FUNCTION_BLOCK ControlDescensoFin
VAR_INPUT
		SFCreset:BOOL;
	    SeguridadOK AT %I*: BOOL;
	    SensorArriba AT %I*: BOOL;
		SensorAbajo AT %I*:BOOL;
		Enabled AT %I*:BOOL;
		PuedeExtraer :BOOL;
		
		SensorPaletDentro AT %I*:BOOL;
		SensorPaletFuera AT %I*:BOOL;
		ElevadorLleno :BOOL;
		PulsadorBajar AT%I*: BOOL;
		PulsadorSubir AT%I*: BOOL;	

		PresenciaCintaArriba AT%I* :BOOL;
		PresenciaCintaAbajo AT %I* : BOOL;	
		
		ResetError :BOOL;
		
		MotorElevacion_Status AT%I*:UINT;
		MotorExtraccion_Status AT%I*:UINT;

END_VAR
VAR_OUTPUT
		MotorElevacion_Freq  AT%Q*: UINT;
	    MotorElevacion_Command AT%Q*: UINT;
		
		MotorExtraccion_Freq  AT%Q*: UINT;
	    MotorExtraccion_Command AT%Q*: UINT;
		
		Ready: BOOL; 
		
END_VAR
VAR
	VelocidadAlta :UINT := 4000;
	VelocidadBAJA :UINT := 1500;
	ModoVelocidadAlta :BOOL := FALSE;
	TiempoAltaVelocidad :TIME := T#3S;
	ERROR :BOOL;
	TimerEntradaSalida: TON;
	
	HomeOK :BOOL;
END_VAR

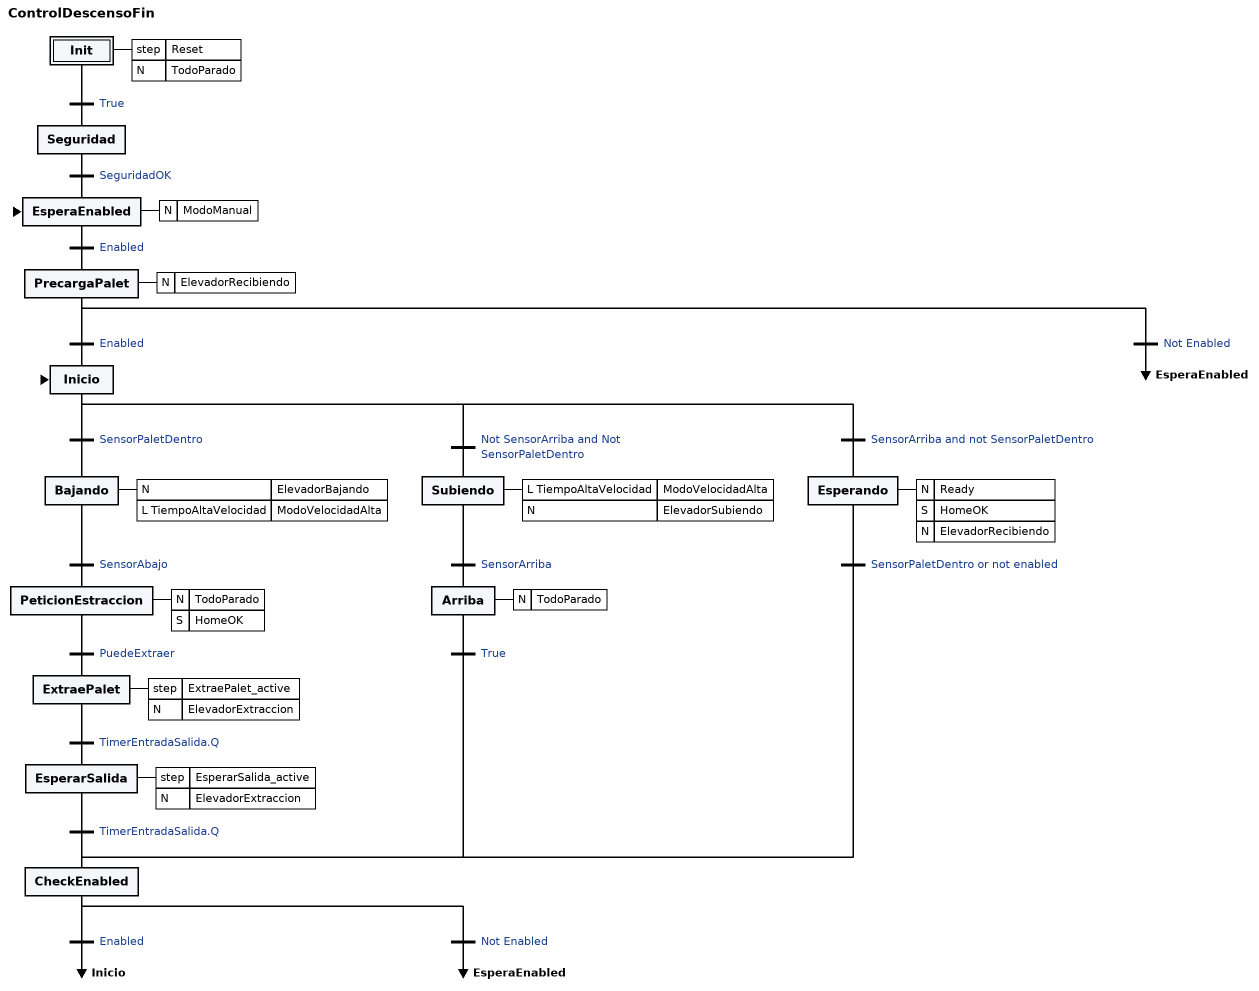
INITIAL_STEP Init:
    Reset(N);  // step action
    TodoParado(N);
END_STEP
TRANSITION FROM Init TO Seguridad
    := True;
END_TRANSITION
STEP Seguridad:
END_STEP
TRANSITION FROM Seguridad TO EsperaEnabled
    := SeguridadOK;
END_TRANSITION
STEP EsperaEnabled:
    ModoManual(N);
END_STEP
TRANSITION FROM EsperaEnabled TO PrecargaPalet
    := Enabled;
END_TRANSITION
STEP PrecargaPalet:  // min time T#2s
    ElevadorRecibiendo(N);
END_STEP
TRANSITION FROM PrecargaPalet TO Inicio
    := Enabled;
END_TRANSITION
TRANSITION FROM PrecargaPalet TO EsperaEnabled
    := Not Enabled;
END_TRANSITION
STEP Inicio:
END_STEP
TRANSITION FROM Inicio TO Bajando
    := SensorPaletDentro;
END_TRANSITION
STEP Bajando:
    ElevadorBajando(N);
    ModoVelocidadAlta(L, TiempoAltaVelocidad);
END_STEP
TRANSITION FROM Bajando TO PeticionEstraccion
    := SensorAbajo;
END_TRANSITION
STEP PeticionEstraccion:
    TodoParado(N);
    HomeOK(S);
END_STEP
TRANSITION FROM PeticionEstraccion TO ExtraePalet
    := PuedeExtraer;
END_TRANSITION
STEP ExtraePalet:  // min time T#1s
    ExtraePalet_active(N);  // step action
    ElevadorExtraccion(N);
END_STEP
TRANSITION FROM ExtraePalet TO EsperarSalida
    := TimerEntradaSalida.Q;
END_TRANSITION
STEP EsperarSalida:
    EsperarSalida_active(N);  // step action
    ElevadorExtraccion(N);
END_STEP
TRANSITION FROM EsperarSalida TO CheckEnabled
    := TimerEntradaSalida.Q;
END_TRANSITION
TRANSITION FROM Inicio TO Subiendo
    := Not SensorArriba and Not SensorPaletDentro;
END_TRANSITION
STEP Subiendo:
    ModoVelocidadAlta(L, TiempoAltaVelocidad);
    ElevadorSubiendo(N);
END_STEP
TRANSITION FROM Subiendo TO Arriba
    := SensorArriba;
END_TRANSITION
STEP Arriba:
    TodoParado(N);
END_STEP
TRANSITION FROM Arriba TO CheckEnabled
    := True;
END_TRANSITION
TRANSITION FROM Inicio TO Esperando
    := SensorArriba and not SensorPaletDentro;
END_TRANSITION
STEP Esperando:
    Ready(N);
    HomeOK(S);
    ElevadorRecibiendo(N);
END_STEP
TRANSITION FROM Esperando TO CheckEnabled
    := SensorPaletDentro or not enabled;
END_TRANSITION
STEP CheckEnabled:
END_STEP
TRANSITION FROM CheckEnabled TO Inicio
    := Enabled;
END_TRANSITION
TRANSITION FROM CheckEnabled TO EsperaEnabled
    := Not Enabled;
END_TRANSITION

ACTION ElevadorBajando:
MotorElevador(2);
MotorExtraccion(0);
END_ACTION

ACTION ElevadorExtraccion:

IF PuedeExtraer THEN
	MotorExtraccion(1);
ELSE 
	MotorExtraccion(0);
END_IF
END_ACTION

ACTION ElevadorRecibiendo:
MotorElevador(0);

IF Enabled THEN
	MotorExtraccion(2);
ELSE 
	MotorExtraccion(0);
END_IF
END_ACTION

ACTION ElevadorSubiendo:
MotorElevador(1);
MotorExtraccion(0);
END_ACTION

ACTION EsperarSalida_active:
TimerEntradaSalida(IN:=NOT PresenciaCintaAbajo, PT:= T#1S);
END_ACTION

ACTION ExtraePalet_active:
TimerEntradaSalida(IN:=PresenciaCintaAbajo, PT:= T#1S);
END_ACTION

ACTION ModoManual:


IF PulsadorSubir THEN
	MotorElevador(1);
		HomeOK :=FALSE;
ELSIF PulsadorBajar THEN
	MotorElevador(2);
		HomeOK :=FALSE;
ELSE
	MotorElevador(0);
END_IF
END_ACTION

METHOD PRIVATE MotorElevador : BOOL
VAR_INPUT
	Direccion : INT; //0 parado 1 subir 2 bajar
END_VAR
IF ModoVelocidadAlta AND HomeOK THEN
	MotorElevacion_Freq := 5000;
ELSE
	MotorElevacion_Freq := 1000;
END_IF


MotorElevacion_Command := 0;
MotorElevacion_Command.7 := 1 ; //Control Word Active

IF Direccion = 0 THEN
	MotorElevacion_Command.3 := 1 ; // Stop according to parameter setting	
ELSIF PresenciaCintaArriba OR PresenciaCintaAbajo THEN
	//ERROR: intenta mover elevador con obstatuclos
	//DEBE MOStrar error
	MotorElevacion_Command.3 := 1 ; // Stop according to parameter setting	
	
ELSIF Direccion  = 1 THEN
		
		MotorElevacion_Command.2 := 0 ; //1 reversed 0 fordward
		MotorElevacion_Command.0 := 1 ; // Run Command active
		HomeOK :=FALSE;

ELSIF Direccion= 2 THEN
	MotorElevacion_Command.2 := 1 ; //1 reversed 0 fordward
	MotorElevacion_Command.0 := 1 ; // Run Command active
		HomeOK :=FALSE;
ELSE
	MotorElevacion_Command.3 := 1 ; // Stop according to parameter setting	
END_IF
END_METHOD

METHOD PRIVATE MotorExtraccion : BOOL
VAR_INPUT
	Direccion : INT; //0 parado 1 salida 2 entrada
END_VAR

MotorExtraccion_Freq := gvl.VelocidadCinta * 100;
MotorExtraccion_Command := 0;
MotorExtraccion_Command.7 := 1 ; //Control Word Active

IF Direccion  = 1 THEN
	MotorExtraccion_Command.2 := 1 ; //1 reversed 0 fordward
	MotorExtraccion_Command.0 := 1 ; // Run Command active
ELSIF Direccion= 2 THEN
	MotorExtraccion_Command.2 := 0 ; //1 reversed 0 fordward
	MotorExtraccion_Command.0 := 1 ; // Run Command active
ELSE
	MotorExtraccion_Command.3 := 1 ; // Stop according to parameter setting	
END_IF
END_METHOD

ACTION RealizaHome:
MotorElevador(1);
MotorExtraccion(0);
END_ACTION

ACTION Reset:
HomeOK := FALSE;
SFCreset:=FALSE;
END_ACTION

ACTION TodoParado:
MotorElevador(0);
MotorExtraccion(0);
END_ACTION

END_FUNCTION_BLOCK

(* stored: Version 1.1.0.1, ProductVersion 3.1.4024.3
   POU ControlDescensoFin: Id {d10a53bb-d051-4ece-977c-1063e3a0bb26}, SpecialFunc None
   Action ElevadorBajando: Id {f417e542-ab0f-4461-b8ce-d469365caa55}
   Action ElevadorExtraccion: Id {226ad220-a433-43f1-9cfa-36101e92e9bd}
   Action ElevadorRecibiendo: Id {b509c615-a273-459a-b38c-2a61db4f1b6a}
   Action ElevadorSubiendo: Id {c1681531-5ba7-4488-b3f6-67dcbabd7920}
   Action EsperarSalida_active: Id {78753ca9-4e77-4c52-b05d-9680293d781a}
   Action ExtraePalet_active: Id {b33e1c20-1db2-43bc-a05c-ff199b115bac}
   Action ModoManual: Id {66938fb8-a4c2-47d6-8638-165a56c0460e}
   Method MotorElevador: Id {da795134-f9f9-4128-900f-470d3e324f12}
   Method MotorExtraccion: Id {f5abc9cf-083f-4ee4-acb4-9a555ffe701e}
   Action RealizaHome: Id {962541b0-be2e-4c0f-b189-25249c8b52b6}
   Action Reset: Id {251a521c-3056-4444-bce8-242a5104f8e6}
   Action TodoParado: Id {59b2797a-5788-4aa8-9401-4e1566db438d} *)
